(* PLC project DuPont_Ultrafiltration_Control, DuPont Ultrafiltration Skid Control 1.0 *)
(* stored: creationDateTime 2023-06-01T12:00:00, modificationDateTime 2023-06-01T12:00:00 *)

PROGRAM UltrafiltrationMain
  VAR
    TON_StateTimer : TON;
    TON_CEBInterval : TON;
    R_TRIG_StartFiltration : R_TRIG;
    R_TRIG_StopSystem : R_TRIG;
    R_TRIG_StartCEB : R_TRIG;
    R_TRIG_StartCIP : R_TRIG;
  END_VAR

            
              INCLUDE "src/POUs/UltrafiltrationMain.st"
            
          
END_PROGRAM

FUNCTION StateIdle

            
              INCLUDE "src/POUs/StateIdle.st"
            
          
END_FUNCTION

FUNCTION StateFiltration

            
              INCLUDE "src/POUs/StateFiltration.st"
            
          
END_FUNCTION

FUNCTION StateAirScour

            
              INCLUDE "src/POUs/StateAirScour.st"
            
          
END_FUNCTION

FUNCTION StateGravityDrain

            
              INCLUDE "src/POUs/StateGravityDrain.st"
            
          
END_FUNCTION

FUNCTION StateBackwashTop

            
              INCLUDE "src/POUs/StateBackwashTop.st"
            
          
END_FUNCTION

FUNCTION StateBackwashBottom

            
              INCLUDE "src/POUs/StateBackwashBottom.st"
            
          
END_FUNCTION

FUNCTION StateForwardFlush

            
              INCLUDE "src/POUs/StateForwardFlush.st"
            
          
END_FUNCTION

FUNCTION_BLOCK StateCEB
  VAR_INPUT
    Start : BOOL;
    Stop : BOOL;
  END_VAR
  VAR_OUTPUT
    Done : BOOL;
    Running : BOOL;
  END_VAR
  VAR
    CEBStep : INT;
    TON_CEBTimer : TON;
  END_VAR

            
              INCLUDE "src/POUs/StateCEB.st"
            
          
END_FUNCTION_BLOCK

FUNCTION_BLOCK StateCIP
  VAR_INPUT
    Start : BOOL;
    Stop : BOOL;
    CIPFilterInstalled : BOOL;
  END_VAR
  VAR_OUTPUT
    Done : BOOL;
    Running : BOOL;
    RequestOperatorConfirmation : BOOL;
    CurrentCIPStep : INT;
    Message : STRING;
  END_VAR
  VAR
    CIPStep : INT;
    TON_CIPTimer : TON;
    CIPInstalled : BOOL;
    SoakTime : time;
    RinseTime : time;
  END_VAR

            
              INCLUDE "src/POUs/StateCIP.st"
            
          
END_FUNCTION_BLOCK

CONFIGURATION DuPont_UF_Config
  RESOURCE PLC_Logic ON PLC
    TASK MainTask(INTERVAL := T#50ms, PRIORITY := 1);
    PROGRAM MainProgram WITH MainTask : UltrafiltrationMain;
  END_RESOURCE
END_CONFIGURATION
